FUNCTION_BLOCK FB_ComponentEX EXTENDS FB_Component
VAR_INPUT
END_VAR
VAR_OUTPUT
END_VAR
VAR
	bAbort:			BOOL;
	bStop:			BOOL;
END_VAR

METHOD PROTECTED M_Execute : BOOL
VAR_INPUT
END_VAR

IF bAbort THEN
	bAbort:= FALSE;
	fbEvent.M_AddSTRING('Test');
	fbEvent.M_AddSTRING('Test2');
	fbEvent.M_AddSTRING('Test3');
	fbEvent.M_Abort('First Error Abort', 'a');
END_IF

IF bStop THEN
	bStop:= FALSE;
	fbEvent.M_AddSTRING('Test');
	fbEvent.M_AddSTRING('Test2');
	fbEvent.M_AddSTRING('Test3');
	fbEvent.M_Stop('First Error Stop', 'b');
END_IF

M_Execute:= True;
END_METHOD

END_FUNCTION_BLOCK

(* stored: Version 1.1.0.1, ProductVersion 3.1.4024.12
   POU FB_ComponentEX: Id {67ecce00-b6ba-4016-865f-4a4dfdc94a76}, SpecialFunc None
   Method M_Execute: Id {bba4d435-5736-45bd-97fd-4ceab6f0d012} *)
